{attribute 'GeneratedUsingTerminal: EL3773-0000-0021'}
{attribute addProperty BoxType "EL3773-0000-0021"}
{attribute addProperty Id "UnderrangeBOOL1OverrangeBOOL1Limit_xBYTE1ErrorBOOL1Sync_errorBOOL1TxPDO_StateBOOL1TxPDO_ToggleBOOL1"}
{attribute addProperty CRC "3700439328"}
{attribute addProperty Size "7"}
TYPE I3_Status_DC903920 :
STRUCT
	{attribute addProperty Name "Underrange"}
	Underrange : BOOL;
	{attribute addProperty Name "Overrange"}
	Overrange : BOOL;
	{attribute addProperty Name "Limit_x"}
	Limit_x : BYTE;
	{attribute addProperty Name "Error"}
	Error : BOOL;
	{attribute addProperty Name "Sync_error"}
	Sync_error : BOOL;
	{attribute addProperty Name "TxPDO_State"}
	TxPDO_State : BOOL;
	{attribute addProperty Name "TxPDO_Toggle"}
	TxPDO_Toggle : BOOL;
END_STRUCT
END_TYPE

(* stored: Version 1.2.0.0, ProductVersion 3.1.4024.11
   DUT I3_Status_DC903920: Id {2777763c-294d-4429-bc31-9e07718b6689} *)
